	REGION CALL_INTERRUPT_CONTINUE
	  // Check for correct interrupt mode
	  CASE #tempInterruptMode OF
	    0, 1: // valid interruptMode
	      #tempInterruptMode := #tempInterruptMode;
	    ELSE
	      // Invalid interruptMode
	      // Use maximum dynamics
	      #tempInterruptMode := 1;
	  END_CASE;

	  #instMC_GroupInterrupt(AxesGroup := #to_Kinematics,
	                         Execute := #statExecGroupInterrupt,
	                         Mode := #tempInterruptMode);

	  // Workaround until FW3.0 -> Interrupt sometimes shows command aborted
	  // Check if interrupt shall be executed and no continue and no stop
	  // Then retrigger interrupt
	  IF #instMC_GroupInterrupt.CommandAborted = TRUE
	    AND #statExecGroupInterrupt = TRUE
	    AND #statExecGroupContinue = FALSE
	    AND #statExecGroupStop = FALSE
	  THEN
	    // Retrigger interrupt
	    #instMC_GroupInterrupt(AxesGroup := #to_Kinematics,
	                           Execute := FALSE,
	                           Mode := #tempInterruptMode);
	    #instMC_GroupInterrupt(AxesGroup := #to_Kinematics,
	                           Execute := TRUE,
	                           Mode := #tempInterruptMode);
	  END_IF;

	  // error detection and signaling
	  IF #instMC_GroupInterrupt.Error THEN
	    #statSubfunctionStatus := #instMC_GroupContinue.ErrorId;
	    #statStatus := #ERR_GROUPINTERRUPT_FAILED; // set status for error evaluation
	  END_IF;



	  #instMC_GroupContinue(AxesGroup := #to_Kinematics,
	                        Execute := #statExecGroupContinue);

	  // error detection and signaling
	  IF #instMC_GroupContinue.Error THEN
	    #statSubfunctionStatus := #instMC_GroupContinue.ErrorId;
	    #statStatus := #ERR_GROUPCONTINUE_FAILED; // set status for error evaluation
	  END_IF;
	END_REGION CALL_INTERRUPT_CONTINUE

	REGION CALL_STOP
	  // Check for correct stop mode
	  CASE #tempStopMode OF
	    0, 1: // normal stopMode
	      #instMC_GroupStop.Mode := #tempStopMode;
	    10: // stopMode with stop of conveyor (path dynamics)
	      #instMC_GroupStop.Mode := 0;
	    11: // stopMode with stop of conveyor (maximum dynamics)
	      #instMC_GroupStop.Mode := 1;
	    ELSE
	      // Invalid stop mode specification
	      // Use maximum dynamics
	      #instMC_GroupStop.Mode := 1;
	  END_CASE;

	  #instMC_GroupStop(AxesGroup := #to_Kinematics,
	                    Execute := #statExecGroupStop);

	  // error detection and signaling
	  IF #instMC_GroupStop.Error THEN
	    #statSubfunctionStatus := #instMC_GroupStop.ErrorId;
	    #statStatus := #ERR_GROUPSTOP_FAILED; // set status for error evaluation
	  END_IF;
	END_REGION CALL_STOP

	REGION CHECK_TO_KINEMATICS_STATE
	  // check TO_Kinematics for pending errors
	  IF #tempKinematicsStatusWord.%X1 = TRUE THEN
	    // only copy statusWords to outputs in case of error
	    #diagnostics.kinematicsStatusWord := #tempKinematicsStatusWord;
	    #diagnostics.kinematicsErrorWord := #tempKinematicsErrorWord;

	    // set status
	    #statStatus := #ERR_TO_KINEMATIC_ERROR;
	  END_IF;

	  // Check if kinematics stopping bit is set but not triggered from here
	  IF #tempKinematicsStatusWord.%X16 = TRUE
	    AND #statStateMachine <> #STOPPING
	    AND #statStateMachine <> #STOPPED_STATE
	    AND #statStateMachine <> #DESYNC_CONVEYOR
	    AND #statStateMachine <> #ERROR_STATE
	    AND #tempStop = FALSE
	  THEN
	    // set bit for detection of external stop
	    #statExternalStopDetected := TRUE;
	    // set state machine
	    #statStateMachine := #STOPPING;
	    #statStatus := #STATUS_PATHMOTION_EXT_STOPPING;
	  END_IF;

	  // Check if conveyor is tracked
	  FOR #tempCtr := 1 TO 3 DO
	    #statActualTrackedOCS := 0;
	    IF #to_Kinematics.StatusConveyor[#tempCtr].TrackingState = 3 THEN
	      #statActualTrackedOCS := DINT_TO_SINT(#tempCtr);
	      EXIT;
	    END_IF;
	  END_FOR;
	END_REGION CHECK_TO_KINEMATICS_STATE

	REGION RESET_ORIENTATION_DYN
	  // change orientation default dynamics back to initial values
	  IF #statOrientationDynChanged THEN
	    #to_Kinematics.DynamicDefaults.Orientation.Velocity := #statOrientationDynOld.velocity;
	    #to_Kinematics.DynamicDefaults.Orientation.Acceleration := #statOrientationDynOld.acceleration;
	    #to_Kinematics.DynamicDefaults.Orientation.Deceleration := #statOrientationDynOld.deceleration;
	    #to_Kinematics.DynamicDefaults.Orientation.Jerk := #statOrientationDynOld.jerk;
	    #statOrientationDynChanged := FALSE;
	  END_IF;
	END_REGION

	REGION OUTPUTS
	  //----------------------------------------------------------------------------------------------
	  // Write ouputs and error handling
	  //----------------------------------------------------------------------------------------------
	  IF (#statStatus.%X15 = TRUE) AND (#statError = FALSE) THEN // Error occurred (#statStatus is 16#8000 to 16#FFFF)
	    #statDone := FALSE;
	    #statBusy := FALSE;
	    #statActive := FALSE;
	    #statCommandAborted := FALSE;
	    #statCmdExecuted := FALSE;
	    #statError := TRUE;
	    #statPauseCmdExecution := FALSE;
	    #statCommandsInExecution := FALSE;
	    // Write diagnostics
	    #diagnostics.stateMachine := #statStateMachine;
	    #diagnostics.status := #statStatus;
	    #diagnostics.motionFBstatus := #statSubfunctionStatus;
	    #statStateMachine := #ERROR_STATE;

	  ELSIF (#statStatus = #STATUS_CMD_EXECUTED) AND (#statDone = FALSE) THEN // command executed to MotionQueue
	    #statDone := FALSE;
	    #statCommandAborted := FALSE;
	    #statError := FALSE;
	    #statCmdExecuted := TRUE;
	    #statStateMachine := #NO_PROCESSING; // Switch state machine to "no processing"

	  ELSIF (#statStatus = #STATUS_PATHMOTION_FINISHED) AND (#statDone = FALSE) THEN // Execution finished without errors
	    #statDone := TRUE;
	    #statBusy := FALSE;
	    #statActive := FALSE;
	    #statCommandAborted := FALSE;
	    #statError := FALSE;
	    #statPauseCmdExecution := FALSE;
	    #statCommandsInExecution := FALSE;
	    #statRemainingDistance := 0.0; // Reset remaining distance when done --> SPTP stays at 1.0, so a reset is necessary
	    #statStateMachine := #NO_PROCESSING; // Switch state machine to "no processing"

	  ELSIF (#statStatus = #STATUS_COMMAND_ABORTED) AND (#statCommandAborted = FALSE) THEN // Commanded functionality has been aborted by another command
	    #statDone := FALSE;
	    #statBusy := FALSE;
	    #statCommandAborted := TRUE;
	    #statError := FALSE;
	    #statCmdExecuted := FALSE;
	    #statPauseCmdExecution := FALSE;
	    #statCommandsInExecution := FALSE;
	    // Write diagnostics
	    #diagnostics.stateMachine := #statStateMachine;
	    #diagnostics.status := #statStatus;
	    #diagnostics.motionFBstatus := #statSubfunctionStatus;
	    #statStateMachine := #NO_PROCESSING; // Switch state machine to "no processing"

	  ELSIF (#tempExecute = FALSE)
	    AND (#tempStop = FALSE)
	    AND (#tempKinematicsStatusWord.%X1 = FALSE) // Avoid toggling statError as kinematics status is checked every cycle
	    AND ((#statDone = TRUE) OR (#statError = TRUE) OR (#statCommandAborted = TRUE))
	  THEN
	    // Reset outputs
	    #statDone := FALSE;
	    #statBusy := FALSE;
	    #statActive := FALSE;
	    #statCommandAborted := FALSE;
	    #statError := FALSE;
	    #statCmdExecuted := FALSE;
	    #statPauseCmdExecution := FALSE;
	    #statCommandsInExecution := FALSE;
	    #statStatus := #STATUS_NO_CALL;
	    // added FR: 2019/04/18 - set state machine to no processing, when ending FB
	    #statStateMachine := #NO_PROCESSING; // Switch state machine to "no processing"
	  END_IF;

	  // Write static values to outputs
	  #done := #statDone;
	  #busy := #statBusy;
	  #active := #statActive;
	  #activeCmdNo := #statActiveCmdNo;
	  #remainingDistanceActCmd := #statRemainingDistance;
	  #pauseCmdExecution := #statPauseCmdExecution;
	  #commandAborted := #statCommandAborted;
	  #error := #statError;
	  #diagnostics.status := #statStatus;
	  #cmdExecuted := #statCmdExecuted;
	  #activeUserFrames := #statActiveUserFrames;
	  #isMeasurementCmd := #statIsMeasurementCmd;


	END_REGION OUTPUTS
	// =================================================================================================================
	// End of Function Block: LKinCtrl_MC_ExecuteKinMotionCmd
	// =================================================================================================================
END_FUNCTION_BLOCK

